Staubli VAL3: type2.dtx

public TrajBigBox box{}
